// TIA Portal V15 export
// export: Created 2018-12-10T18:36:39.5512674Z, ExportSetting WithDefaults, WithReadOnly, DisplayName Totally Integrated Automation Portal, DisplayVersion V15 Update 2, DisplayName TIA Portal Openness, DisplayVersion V15 Update 2, DisplayName STEP 7 Professional, DisplayVersion V15 Update 2, DisplayName STEP 7 Safety, DisplayVersion V15, DisplayName WinCC Professional, DisplayVersion V15 Update 2, DisplayName SIMATIC Visualization Architect, DisplayVersion V15 Update 1
DATA_BLOCK "FGDB_ROBNAME@Riveting"   // DB95
TITLE = Technology riveting / Technologie Nieten
{ S7_Optimized_Access := 'FALSE' }
AUTHOR : integra
FAMILY : SUB
VERSION : 0.1
// stored: AutoNumber true, CodeModifiedDate 2018-02-20T07:54:55.2995227Z, CompileDate 2018-02-20T10:24:48.0332036Z, CreationDate 2017-02-23T09:16:27.5672042Z, DBAccessibleFromOPCUA true, InstanceOfName iSF_TECH_ROBOT_RIVETING, InstanceOfNumber 43, InstanceOfType FB, InterfaceModifiedDate 2018-02-19T12:46:15.5811037Z, IsConsistent true, IsKnowHowProtected false, ModifiedDate 2018-02-20T07:54:55.2995227Z, ParameterModified 2018-02-19T12:44:53.8839037Z, StructureModified 2018-02-19T12:46:15.5811037Z, UDAEnableTagReadback false
"iSF_TECH_ROBOT_RIVETING"
   // VAR_INPUT
   //    fct : Int;
   //    safetyStop : Bool;
   //    functionPoint : String[6];
   //    identType : String[12];
   // END_VAR
   // VAR_OUTPUT
   //    counterParts : Int;
   //    counterNIOpoints : Int;
   //    counterIOpoints : Int;
   //    fault : Bool;
   // END_VAR
   // VAR_IN_OUT
   //    IfcFGExternal : "iUDT_IFC_SYS_EXTERNAL_ALARM";
   //    IfcTECH : "iUDT_IFC_ROBOT_TECH";
   //    IfcAcyclicdata : "iUDT_IFC_ROBOT_ACYCLICDATA";
   //    ident : Variant;
   //    IfcTLG : "iUDT_IFC_TLG";
   //    TLG_MQDV : "iUDT_TLG_MQDV_ROBOT";
   //    TLG_ENEV : "iUDT_TLG_ENEV";
   //    In_PI_TECH : "iUDT_PI_ROBOT_ADRxx48_TECH";
   //    Out_PO_TECH : "iUDT_PO_ROBOT_ADRxx48_TECH";
   // END_VAR
   // VAR RETAIN
   //    F : Struct
   //       wrongID : Bool;
   //       notReady : Bool;
   //       Controllerfault : Bool;
   //       processStop : Bool;
   //       toolcheckNIO : Bool;
   //       plus : Bool;
   //    END_STRUCT;
   //    W : Struct
   //       processError : Bool;
   //       maintenanceReq : Bool;
   //       warningLimit : Bool;
   //       quantityMAX : Bool;
   //       teaching : Bool;
   //       processMonitoring : Bool;
   //       rivetLengthControl : Bool;
   //       rivetSeparater : Bool;
   //       limitRivet_A : Bool;
   //       limitRivet_B : Bool;
   //       connectionHMI : Bool;
   //    END_STRUCT;
   //    Masks : Struct
   //       disableFault1_8 : Byte;
   //       prodRelevantFault1_8 : Byte;
   //       prodRelevantWarningt_1_8 : Byte;
   //       prodRelevantWarningt_9_16 : Byte;
   //    END_STRUCT;
   //    LastState : Struct
   //       fault1_8 : Byte;
   //       warning_1_8 : Byte;
   //       warning_9_16 : Byte;
   //    END_STRUCT;
   //    Tmr : Struct
   //       s1 { S7_SetPoint := 'True'} : Int;
   //       a1 : Int;
   //    END_STRUCT;
   //    TmrB : Struct
   //       "1_EnableDelayTime" : Bool;
   //       "1_RunDelayTime" : Bool;
   //       "1_DoneDelayTime" : Bool;
   //    END_STRUCT;
   //    TECH : Struct
   //       ID : Byte;
   //       ready : Bool;
   //       automaticActive : Bool;
   //       qualityNOK : Bool;
   //       qualityOK : Bool;
   //       processError : Bool;
   //       controllerFault : Bool;
   //       processStop : Bool;
   //       maintenanceReq : Bool;
   //       toolcheckNIO : Bool;
   //       warningLimit : Bool;
   //       quantityMAx : Bool;
   //       activeSTO : Bool;
   //       activeTeaching : Bool;
   //       processMonitoring : Bool;
   //       activeOperatorprotection : Bool;
   //       activeRivetLengthControl : Bool;
   //       confirmAccess : Bool;
   //       rivetSeparater : Bool;
   //       limitRivet_A : Bool;
   //       limitRivet_B : Bool;
   //       connectionHMI : Bool;
   //       technoBit22 : Bool;
   //       technoBit23 : Bool;
   //       technoBit24 : Bool;
   //       technoBit25 : Bool;
   //       technoBit26 : Bool;
   //       technoBit27 : Bool;
   //       technoBit28 : Bool;
   //       technoBit29 : Bool;
   //       technoBit30 : Bool;
   //       technoBit31 : Bool;
   //       technoBit32 : Bool;
   //       technoBit33 : Bool;
   //       technoBit34 : Bool;
   //       technoBit35 : Bool;
   //       technoBit36 : Bool;
   //       technoBit37 : Bool;
   //       technoBit38 : Bool;
   //       technoBit39 : Bool;
   //       technoBit40 : Bool;
   //    END_STRUCT;
   //    PLUS : "iIF_ROBOT_PLUS";
   // END_VAR
BEGIN
END_DATA_BLOCK
